Xinje XCPPro project, PLC1: XC3-24 (software 3.3k)

PROGRAM Ladder

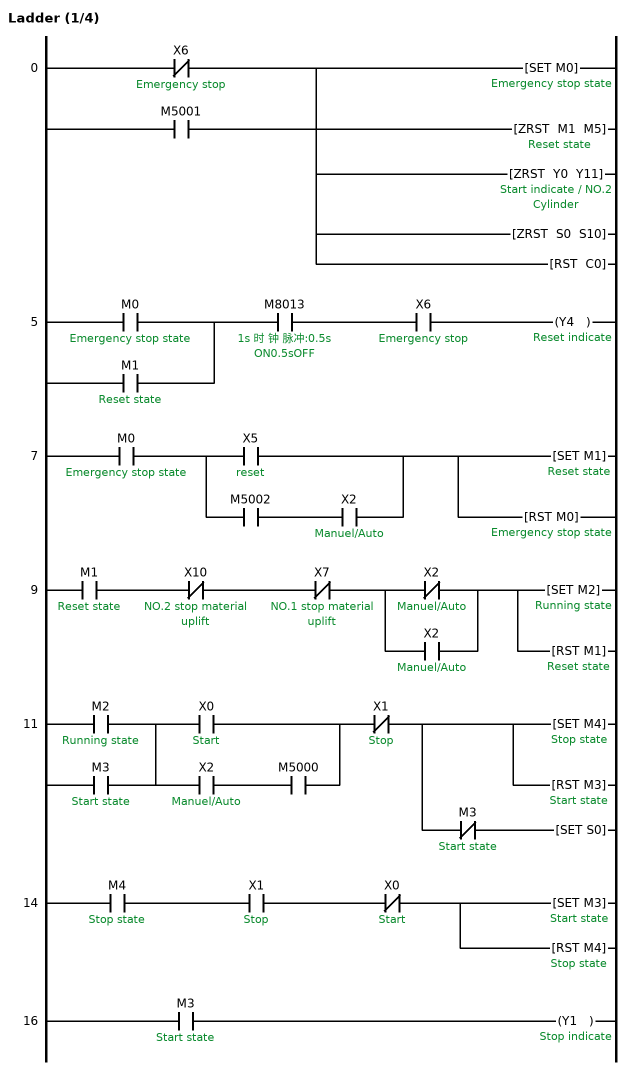
LDI    X6	; Emergency stop
OR     M5001
SET    M0	; Emergency stop state
ZRST   M1 M5	; Reset state
ZRST   Y0 Y11	; Start indicate / NO.2 Cylinder
ZRST   S0 S10
RST    C0
LD     M0	; Emergency stop state
OR     M1	; Reset state
AND    M8013	; 1s 时 钟 脉冲:0.5s ON0.5sOFF
AND    X6	; Emergency stop
OUT    Y4	; Reset indicate
LD     M0	; Emergency stop state
LD     X5	; reset
LD     M5002
AND    X2	; Manuel/Auto
ORB
ANB
SET    M1	; Reset state
RST    M0	; Emergency stop state
LD     M1	; Reset state
ANI    X10	; NO.2 stop material uplift
ANI    X7	; NO.1 stop material uplift
LDI    X2	; Manuel/Auto
OR     X2	; Manuel/Auto
ANB
SET    M2	; Running state
RST    M1	; Reset state
LD     M2	; Running state
OR     M3	; Start state
LD     X0	; Start
LD     X2	; Manuel/Auto
AND    M5000
ORB
ANB
ANI    X1	; Stop
SET    M4	; Stop state
RST    M3	; Start state
ANI    M3	; Start state
SET    S0
LD     M4	; Stop state
AND    X1	; Stop
ANI    X0	; Start
SET    M3	; Start state
RST    M4	; Stop state
LD     M3	; Start state
OUT    Y1	; Stop indicate

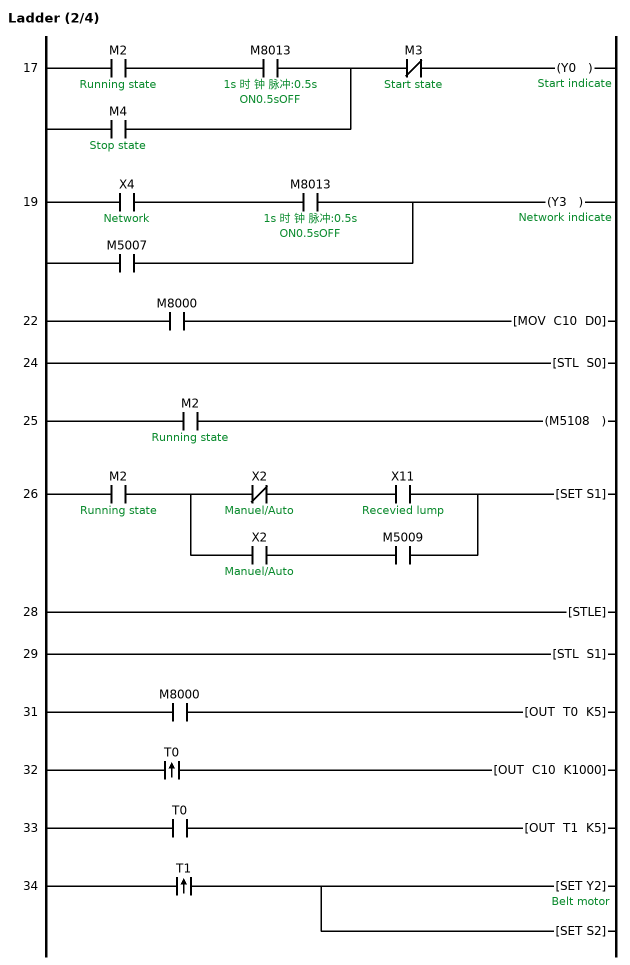
LD     M2	; Running state
AND    M8013	; 1s 时 钟 脉冲:0.5s ON0.5sOFF
OR     M4	; Stop state
ANI    M3	; Start state
OUT    Y0	; Start indicate
LD     X4	; Network
AND    M8013	; 1s 时 钟 脉冲:0.5s ON0.5sOFF
OR     M5007
OUT    Y3	; Network indicate
LD     M8000
MOV    C10 D0
STL    S0
LD     M2	; Running state
OUT    M5108
LD     M2	; Running state
LDI    X2	; Manuel/Auto
AND    X11	; Recevied lump
LD     X2	; Manuel/Auto
AND    M5009
ORB
ANB
SET    S1
STLE
STL    S1
LD     M8000
OUT    T0 K5
LDP    T0
OUT    C10 K1000
LD     T0
OUT    T1 K5
LDP    T1
SET    Y2	; Belt motor
SET    S2

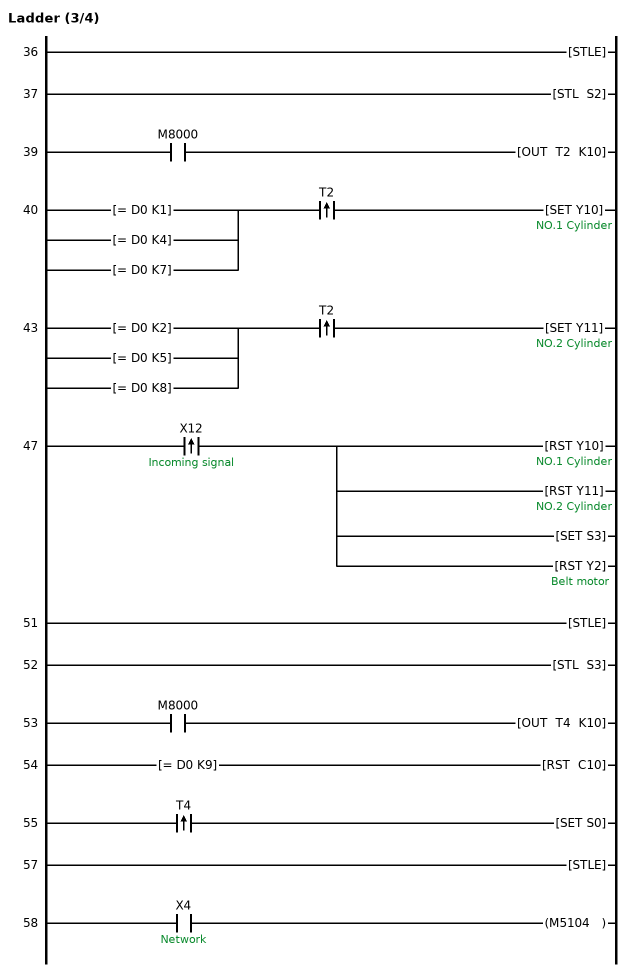
STLE
STL    S2
LD     M8000
OUT    T2 K10
LD=    D0 K1
OR=    D0 K4
OR=    D0 K7
ANDP   T2
SET    Y10	; NO.1 Cylinder
LD=    D0 K2
OR=    D0 K5
OR=    D0 K8
ANDP   T2
SET    Y11	; NO.2 Cylinder
LDP    X12	; Incoming signal
RST    Y10	; NO.1 Cylinder
RST    Y11	; NO.2 Cylinder
SET    S3
RST    Y2	; Belt motor
STLE
STL    S3
LD     M8000
OUT    T4 K10
LD=    D0 K9
RST    C10
LDP    T4
SET    S0
STLE
LD     X4	; Network
OUT    M5104

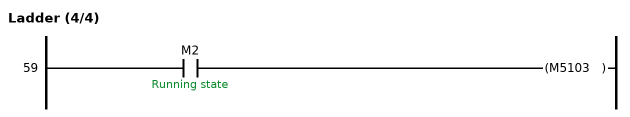
LD     M2	; Running state
OUT    M5103

COMMENTS (devices not used above)
Y5	Alarm indicate